(* PLC project Beremiz non-standard POUs library, Beremiz Beremiz 0.0 *)
(* stored: creationDateTime 2008-12-14T16:53:26, modificationDateTime 2025-02-03T14:57:54 *)

(* Triggers CSV read FB to refresh output, without reloading CSV files *)
FUNCTION_BLOCK csv_refresh
  VAR_EXTERNAL
    pyext_csv_update : INT;
  END_VAR
  VAR_INPUT
    TRIG : BOOL;
  END_VAR
  VAR  (* added by the conversion: wires and edge detectors of the diagram *)
    R_TRIG1 : R_TRIG;
    _ADD13_ENO : BOOL;
    _ADD13_OUT : INT;
  END_VAR

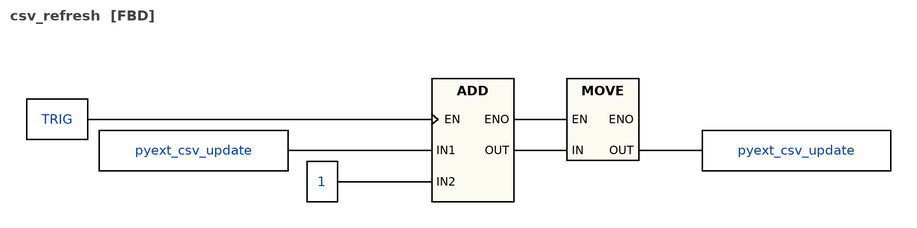
(* FBD diagram, written out as Structured Text *)
R_TRIG1(CLK := TRIG);
_ADD13_OUT := ADD(EN := R_TRIG1.Q, IN1 := pyext_csv_update, IN2 := 1, ENO => _ADD13_ENO);
IF _ADD13_ENO THEN pyext_csv_update := _ADD13_OUT; END_IF;
END_FUNCTION_BLOCK

FUNCTION_BLOCK python_eval
  VAR_INPUT
    TRIG : BOOL;
    CODE : STRING;
  END_VAR
  VAR_OUTPUT
    ACK : BOOL;
    RESULT : STRING;
  END_VAR
  VAR
    STATE : DWORD;
    BUFFER : STRING;
    PREBUFFER : STRING;
    TRIGM1 : BOOL;
    TRIGGED : BOOL;
    SLOT : DINT;  (* Index of this instance's entry in the eval fifo, while a request is in flight. A logic hot-swap stores ~index instead, until the instance the PLC runs claims that entry back. *)
  END_VAR

            {extern void __PythonEvalFB(int, PYTHON_EVAL_data__*);__PythonEvalFB(0, data__);}
          
END_FUNCTION_BLOCK

FUNCTION_BLOCK csv_write_by_string
  VAR_OUTPUT
    ACK : BOOL;
    ERROR : BOOL;
    RESULT : STRING;
  END_VAR
  VAR_INPUT
    FILE_NAME : STRING;
    ROW : STRING;
    COLUMN : STRING;
    CONTENT : STRING;
    SAVE : BOOL;
  END_VAR
  VAR
    py_eval0 : python_eval;
    R_TRIG1 : R_TRIG;
    R_TRIG2 : R_TRIG;
    csv_refresh0 : csv_refresh;
  END_VAR
  VAR  (* added by the conversion: wires and edge detectors of the diagram *)
    _EQ34_OUT : BOOL;
  END_VAR

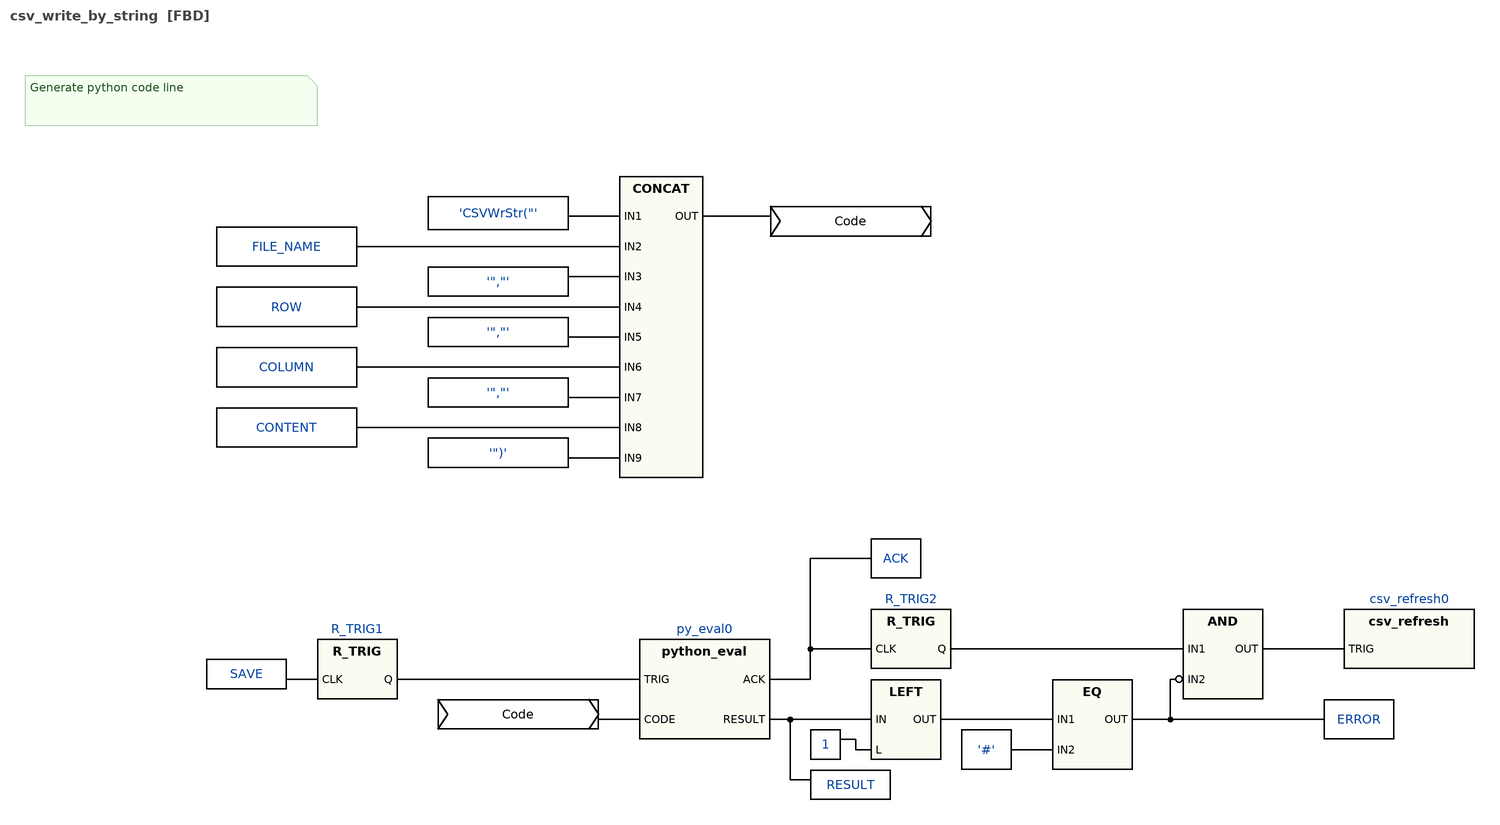
(* FBD diagram, written out as Structured Text *)
(* Generate python code line *)
R_TRIG1(CLK := SAVE);
py_eval0(TRIG := R_TRIG1.Q, CODE := CONCAT('CSVWrStr("', FILE_NAME, '","', ROW, '","', COLUMN, '","', CONTENT, '")'));
ACK := py_eval0.ACK;
_EQ34_OUT := LEFT(py_eval0.RESULT, 1) = '#';
ERROR := _EQ34_OUT;
RESULT := py_eval0.RESULT;
R_TRIG2(CLK := py_eval0.ACK);
csv_refresh0(TRIG := R_TRIG2.Q AND NOT _EQ34_OUT);
END_FUNCTION_BLOCK

FUNCTION_BLOCK _csv_update
  VAR_EXTERNAL
    pyext_csv_update : INT;
  END_VAR
  VAR
    pyext_csv_update_tmp : INT;
  END_VAR
  VAR_OUTPUT
    TRIG : BOOL;
  END_VAR
  VAR
    R_TRIG0 : R_TRIG;
  END_VAR

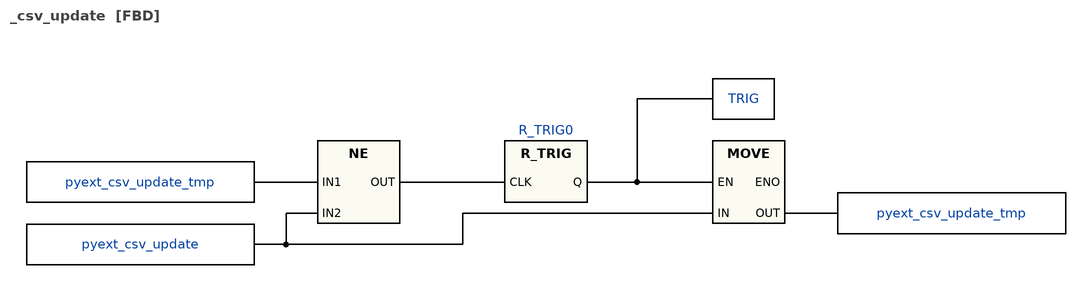
(* FBD diagram, written out as Structured Text *)
R_TRIG0(CLK := pyext_csv_update_tmp <> pyext_csv_update);
TRIG := R_TRIG0.Q;
IF R_TRIG0.Q THEN pyext_csv_update_tmp := pyext_csv_update; END_IF;
END_FUNCTION_BLOCK

FUNCTION_BLOCK csv_read_by_string
  VAR_OUTPUT
    ACK : BOOL;
    RESULT : STRING;
  END_VAR
  VAR_INPUT
    FILE_NAME : STRING;
    ROW : STRING;
    COLUMN : STRING;
  END_VAR
  VAR
    OLDCODE : STRING;
    py_eval : python_eval;
    R_TRIG1 : R_TRIG;
    SR0 : SR;
    _csv_update0 : _csv_update;
  END_VAR
  VAR  (* added by the conversion: wires and edge detectors of the diagram *)
    _OR15_OUT : BOOL;
    R_TRIG1_2 : R_TRIG;
  END_VAR

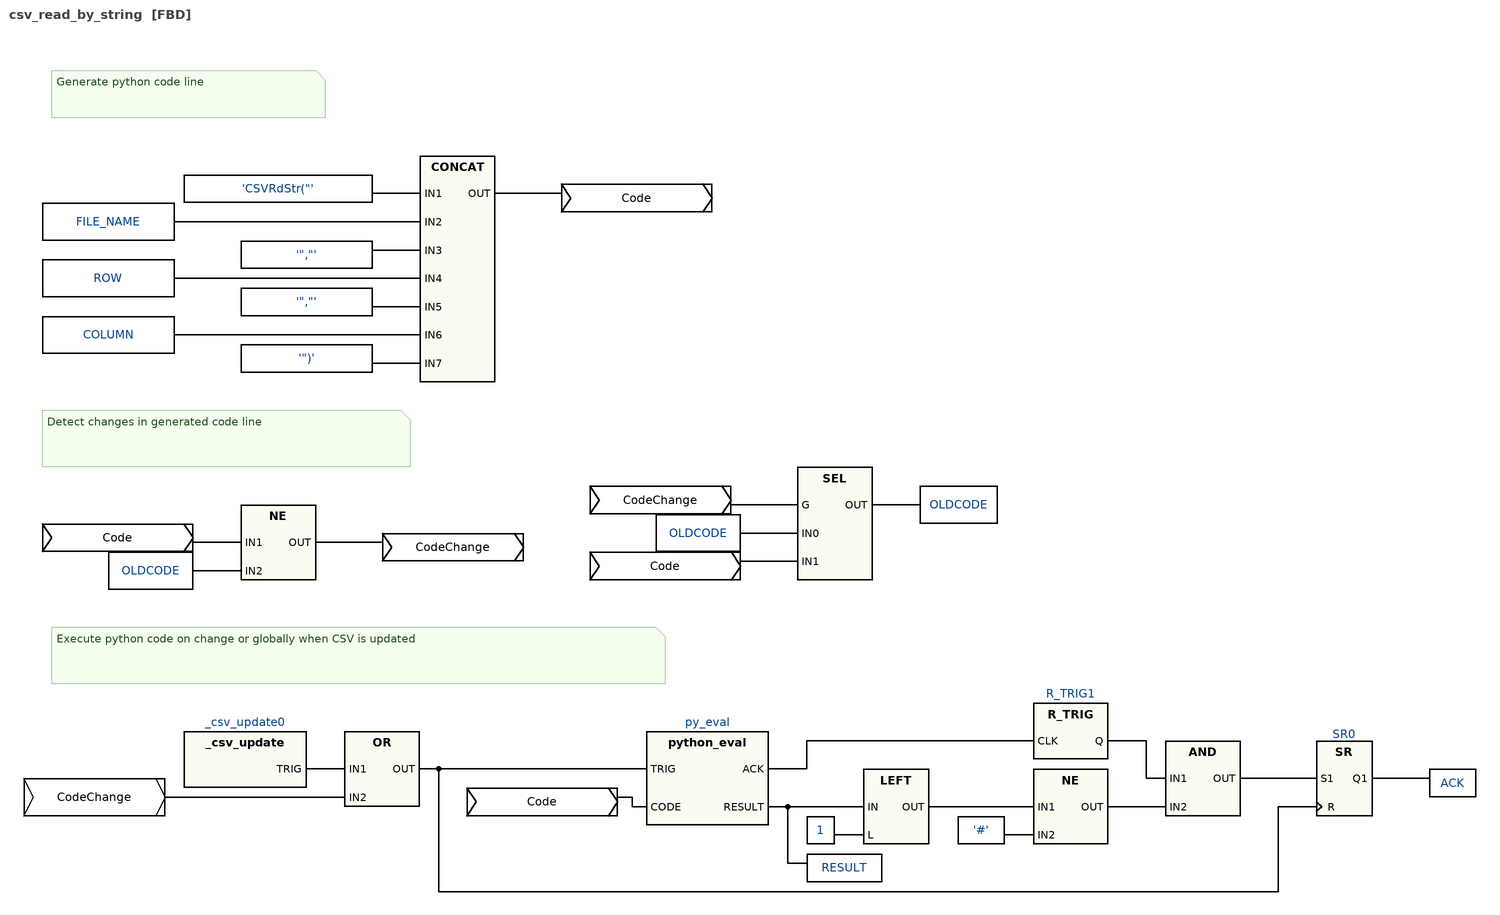
(* FBD diagram, written out as Structured Text *)
(* Generate python code line *)
(* Detect changes in generated code line *)
OLDCODE := SEL(CONCAT('CSVRdStr("', FILE_NAME, '","', ROW, '","', COLUMN, '")') <> OLDCODE, OLDCODE, CONCAT('CSVRdStr("', FILE_NAME, '","', ROW, '","', COLUMN, '")'));
(* Execute python code on change or globally when CSV is updated *)
_csv_update0();
_OR15_OUT := _csv_update0.TRIG OR CONCAT('CSVRdStr("', FILE_NAME, '","', ROW, '","', COLUMN, '")') <> OLDCODE;
py_eval(TRIG := _OR15_OUT, CODE := CONCAT('CSVRdStr("', FILE_NAME, '","', ROW, '","', COLUMN, '")'));
R_TRIG1(CLK := py_eval.ACK);
R_TRIG1_2(CLK := _OR15_OUT);
SR0(S1 := R_TRIG1.Q AND LEFT(py_eval.RESULT, 1) <> '#', R := R_TRIG1_2.Q);
ACK := SR0.Q1;
RESULT := py_eval.RESULT;
END_FUNCTION_BLOCK

(* Purge CSV files cache and refresh CSV read FBs outputs, consequently reloading CSV files *)
FUNCTION_BLOCK csv_reload
  VAR_OUTPUT
    ACK : BOOL;
    RESULT : STRING;
  END_VAR
  VAR
    py_eval : python_eval;
  END_VAR
  VAR_INPUT
    TRIG : BOOL;
  END_VAR
  VAR
    csv_refresh0 : csv_refresh;
  END_VAR

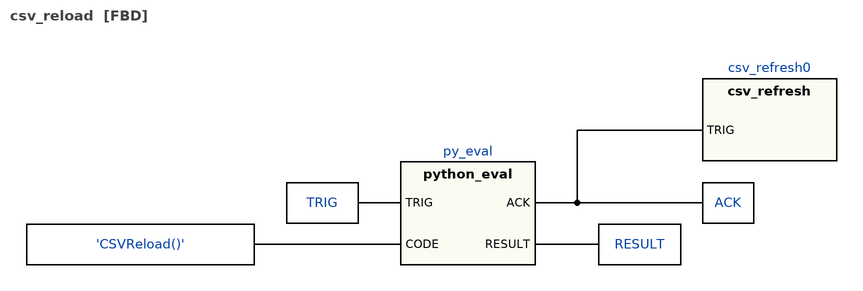
(* FBD diagram, written out as Structured Text *)
py_eval(TRIG := TRIG, CODE := 'CSVReload()');
ACK := py_eval.ACK;
RESULT := py_eval.RESULT;
csv_refresh0(TRIG := py_eval.ACK);
END_FUNCTION_BLOCK

FUNCTION_BLOCK csv_read_by_int
  VAR_OUTPUT
    ACK : BOOL;
    RESULT : STRING;
  END_VAR
  VAR_INPUT
    FILE_NAME : STRING;
    ROW : INT;
    COLUMN : INT;
  END_VAR
  VAR
    OLDCODE : STRING;
    py_eval0 : python_eval;
    R_TRIG2 : R_TRIG;
    SR0 : SR;
    _csv_update0 : _csv_update;
  END_VAR
  VAR  (* added by the conversion: wires and edge detectors of the diagram *)
    _OR15_OUT : BOOL;
    R_TRIG1 : R_TRIG;
  END_VAR

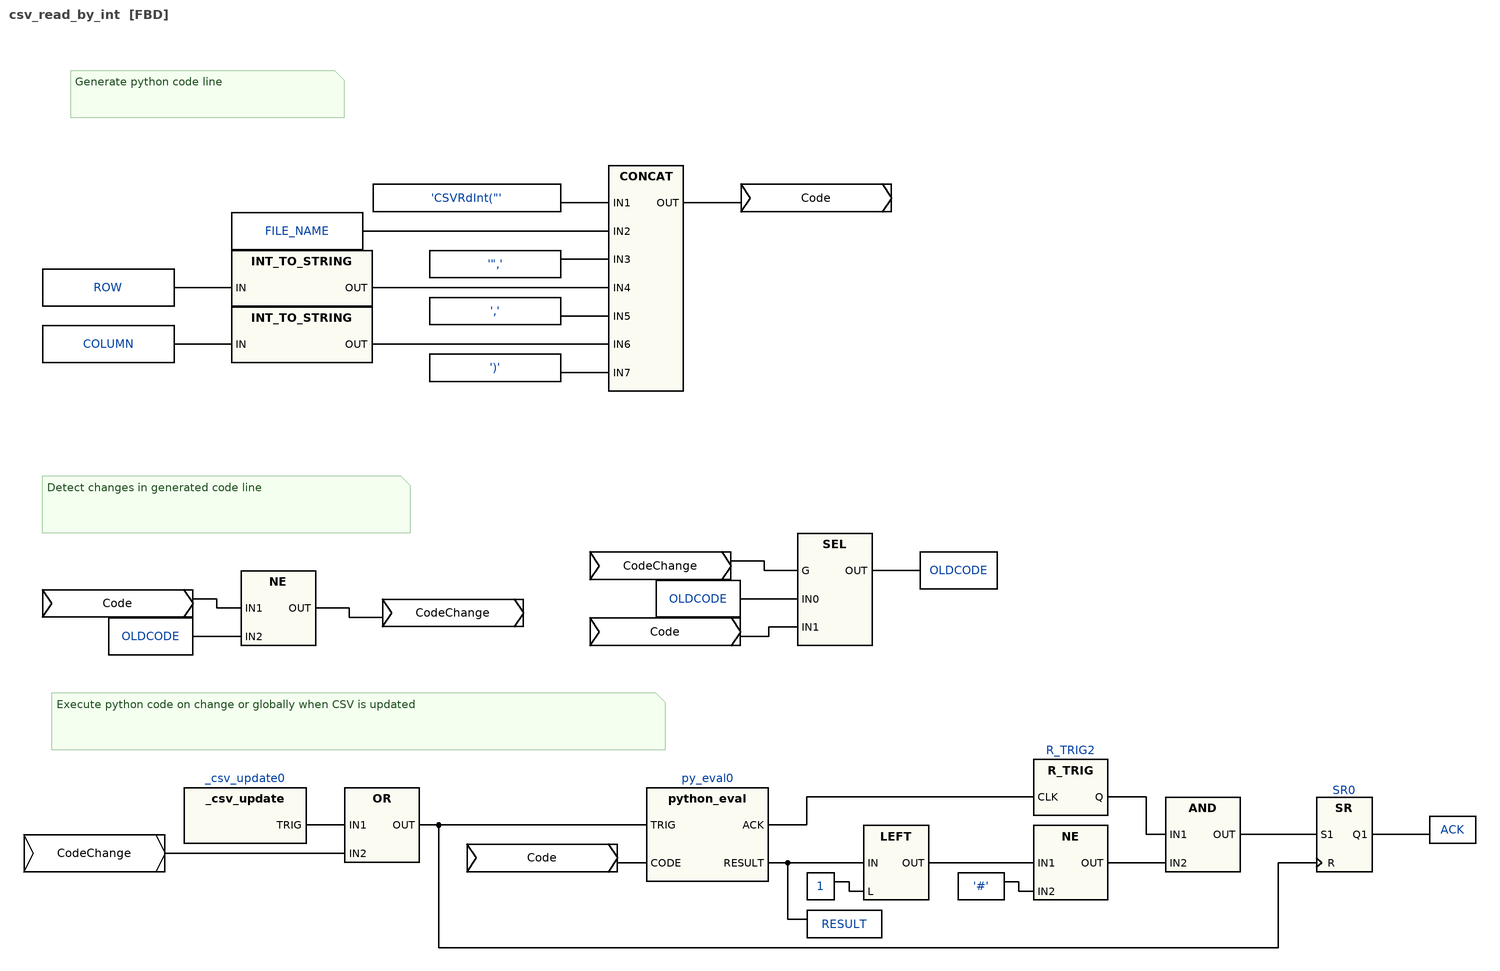
(* FBD diagram, written out as Structured Text *)
(* Generate python code line *)
(* Detect changes in generated code line *)
OLDCODE := SEL(CONCAT('CSVRdInt("', FILE_NAME, '",', INT_TO_STRING(ROW), ',', INT_TO_STRING(COLUMN), ')') <> OLDCODE, OLDCODE, CONCAT('CSVRdInt("', FILE_NAME, '",', INT_TO_STRING(ROW), ',', INT_TO_STRING(COLUMN), ')'));
(* Execute python code on change or globally when CSV is updated *)
_csv_update0();
_OR15_OUT := _csv_update0.TRIG OR CONCAT('CSVRdInt("', FILE_NAME, '",', INT_TO_STRING(ROW), ',', INT_TO_STRING(COLUMN), ')') <> OLDCODE;
py_eval0(TRIG := _OR15_OUT, CODE := CONCAT('CSVRdInt("', FILE_NAME, '",', INT_TO_STRING(ROW), ',', INT_TO_STRING(COLUMN), ')'));
R_TRIG2(CLK := py_eval0.ACK);
R_TRIG1(CLK := _OR15_OUT);
SR0(S1 := R_TRIG2.Q AND LEFT(py_eval0.RESULT, 1) <> '#', R := R_TRIG1.Q);
ACK := SR0.Q1;
RESULT := py_eval0.RESULT;
END_FUNCTION_BLOCK

FUNCTION_BLOCK csv_write_by_int
  VAR_OUTPUT
    ACK : BOOL;
    ERROR : BOOL;
    RESULT : STRING;
  END_VAR
  VAR_INPUT
    FILE_NAME : STRING;
    ROW : INT;
    COLUMN : INT;
    CONTENT : STRING;
    SAVE : BOOL;
  END_VAR
  VAR
    py_eval0 : python_eval;
    R_TRIG1 : R_TRIG;
    R_TRIG2 : R_TRIG;
    csv_refresh0 : csv_refresh;
  END_VAR
  VAR  (* added by the conversion: wires and edge detectors of the diagram *)
    _EQ34_OUT : BOOL;
  END_VAR

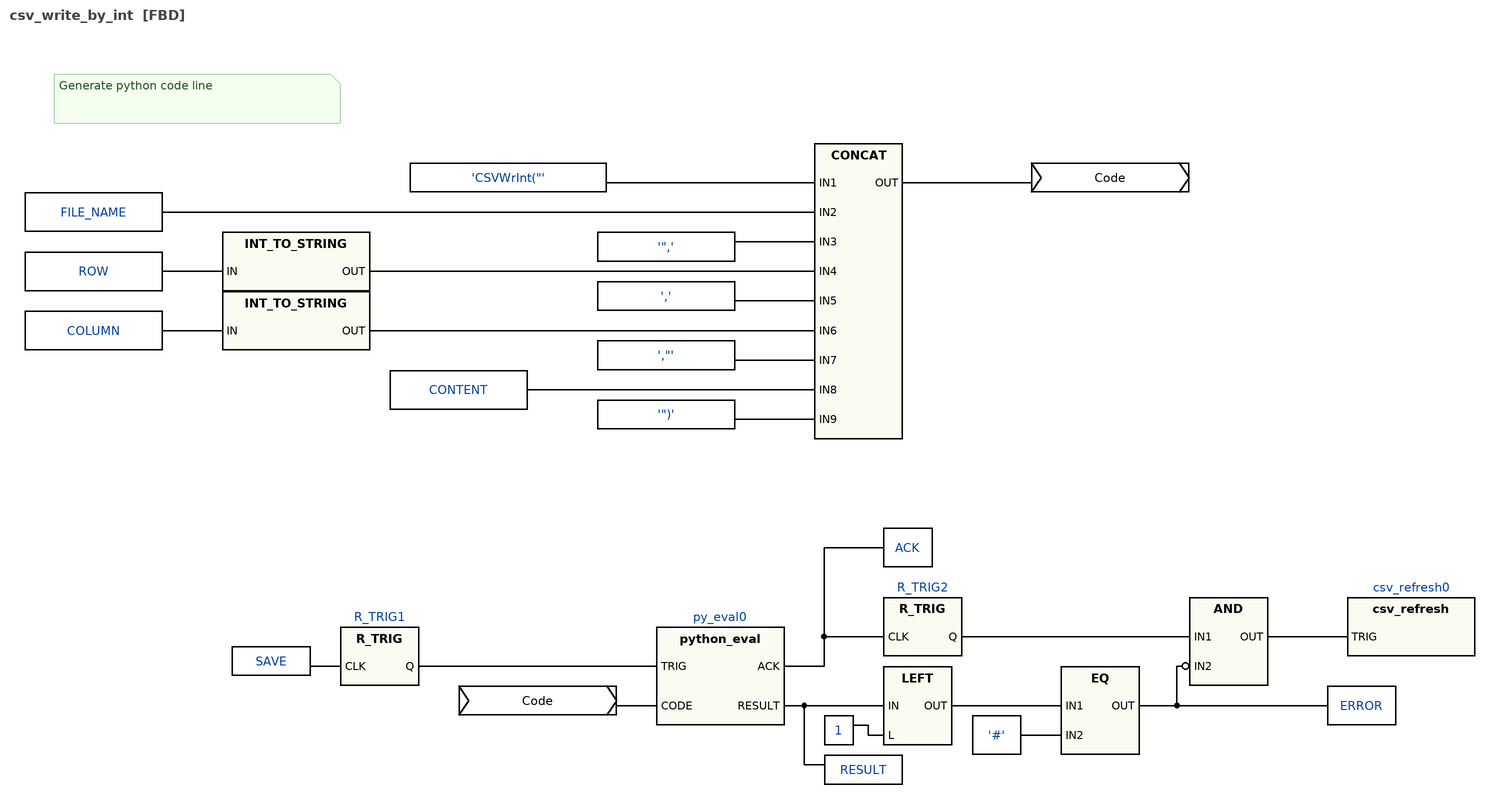
(* FBD diagram, written out as Structured Text *)
(* Generate python code line *)
R_TRIG1(CLK := SAVE);
py_eval0(TRIG := R_TRIG1.Q, CODE := CONCAT('CSVWrInt("', FILE_NAME, '",', INT_TO_STRING(ROW), ',', INT_TO_STRING(COLUMN), ',"', CONTENT, '")'));
ACK := py_eval0.ACK;
_EQ34_OUT := LEFT(py_eval0.RESULT, 1) = '#';
ERROR := _EQ34_OUT;
RESULT := py_eval0.RESULT;
R_TRIG2(CLK := py_eval0.ACK);
csv_refresh0(TRIG := R_TRIG2.Q AND NOT _EQ34_OUT);
END_FUNCTION_BLOCK

FUNCTION_BLOCK python_poll
  VAR_INPUT
    TRIG : BOOL;
    CODE : STRING;
  END_VAR
  VAR_OUTPUT
    ACK : BOOL;
    RESULT : STRING;
  END_VAR
  VAR
    STATE : DWORD;
    BUFFER : STRING;
    PREBUFFER : STRING;
    TRIGM1 : BOOL;
    TRIGGED : BOOL;
    SLOT : DINT;  (* Index of this instance's entry in the eval fifo, while a request is in flight. A logic hot-swap stores ~index instead, until the instance the PLC runs claims that entry back. *)
  END_VAR

            {extern void __PythonEvalFB(int, PYTHON_EVAL_data__*);__PythonEvalFB(1,(PYTHON_EVAL_data__*)(void*)data__);}
          
END_FUNCTION_BLOCK

FUNCTION_BLOCK python_gear
  VAR_INPUT
    N : UINT;
    TRIG : BOOL;
    CODE : STRING;
  END_VAR
  VAR_OUTPUT
    ACK : BOOL;
    RESULT : STRING;
  END_VAR
  VAR
    py_eval : python_eval;
    COUNTER : UINT;
  END_VAR
  VAR  (* added by the conversion: wires and edge detectors of the diagram *)
    _ADD10_OUT : UINT;
    _EQ13_OUT : BOOL;
  END_VAR

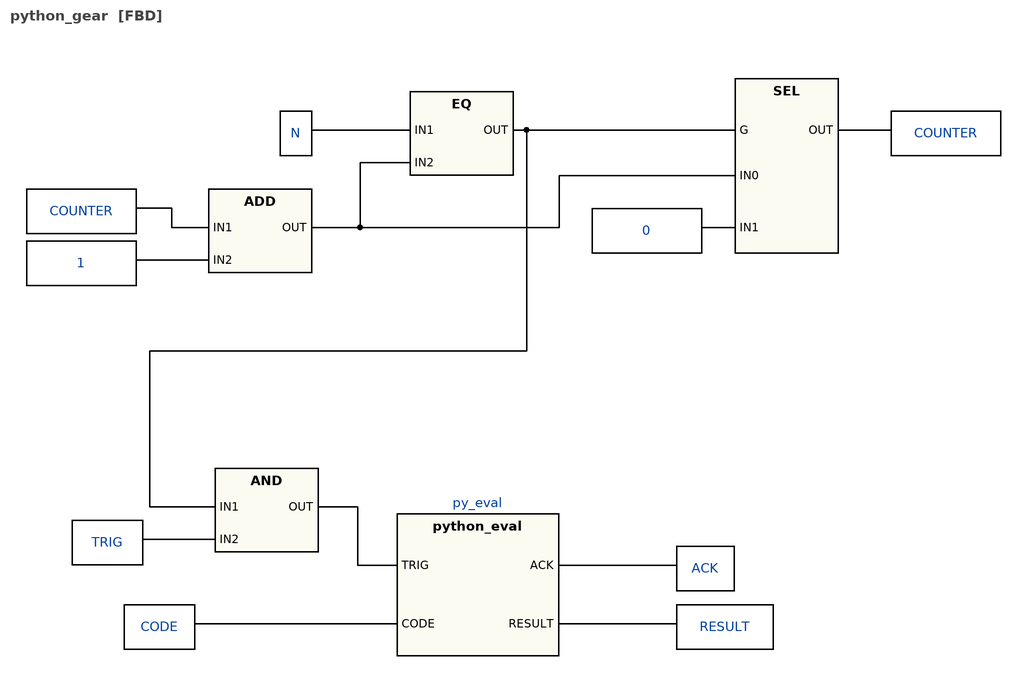
(* FBD diagram, written out as Structured Text *)
_ADD10_OUT := COUNTER + 1;
_EQ13_OUT := N = _ADD10_OUT;
COUNTER := SEL(_EQ13_OUT, _ADD10_OUT, 0);
py_eval(TRIG := _EQ13_OUT AND TRIG, CODE := CODE);
ACK := py_eval.ACK;
RESULT := py_eval.RESULT;
END_FUNCTION_BLOCK

CONFIGURATION configuration0
  VAR_GLOBAL
    pyext_csv_update : INT := 0;
  END_VAR
END_CONFIGURATION
